// TIA Portal V18 export
VAR_GLOBAL   // PLC tag table "04_9 Costanti Nomi Attuatore Stz09"
END_VAR
VAR_GLOBAL CONSTANT   // user constants
   M401 : Int := 1;   // Motore carro tagli
   M404 : Int := 2;   // Motore salita/discesa disco
   M405 : Int := 3;   // Motore rotazione disco
   M408 : Int := 4;   // Motore tappeto evacuazione
   P901 : Int := 5;   // EV pressore profilo
   P902 : Int := 6;   // EV morse ingresso
   P903 : Int := 7;   // EV morse uscita
END_VAR
